(* PLC project x *)

PROGRAM FBD_EMPTY
  VAR
    x : BOOL;
  END_VAR

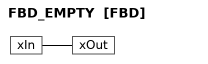
(* FBD diagram, written out as Structured Text *)
(* // Section header: E-STOP CHAIN (documentation-only network) *)
(* --- network: Title of network one --- *)
(* // second network comment *)
(* --- network: Title of network two --- *)
xOut := xIn;
END_PROGRAM
